PROGRAM MAIN
VAR
END_VAR

RunGrindingWheel();

END_PROGRAM

(* stored: Version 1.1.0.1, ProductVersion 3.1.4024.6
   POU MAIN: Id {60175d8f-0214-4e23-95d0-d4930708b4e9}, SpecialFunc None *)
